{attribute addProperty BoxType "EK1122-0000-0018"}
{attribute addProperty Id "Beckhoff_EKM1xxxsub_EK1100EK1100_179A0949162A_0001_EKM1101_0000_0016EKM1101_87969BFD51464.25A_0002_EKM1101_0000_0017EKM1101_87969BFD51464.25A_0003_EKM1101_0000_0018EKM1101_87969BFD51464.25A_0004_EKM1101_0000_0019EKM1101_87969BFD51464.25A_0005_EKM1101_0000_0020EKM1101_87969BFD51464.25"}
{attribute addProperty CRC "2110049489"}
{attribute addProperty SizeInBites "2586"}
{attribute addProperty SizeInBytes "323.25"}
TYPE Beckhoff_EKM1xxxEK1122_7DC4CCD1 EXTENDS EK1122_179A0949 :
STRUCT
	{attribute addProperty Name "Beckhoff_EKM1xxxsub_EK1100"}
	Beckhoff_EKM1xxxsub_EK1100 : EK1100_179A0949;
	{attribute addProperty Name "A_0001_EKM1101_0000_0016"}
	A_0001_EKM1101_0000_0016 : EKM1101_87969BFD;
	{attribute addProperty Name "A_0002_EKM1101_0000_0017"}
	A_0002_EKM1101_0000_0017 : EKM1101_87969BFD;
	{attribute addProperty Name "A_0003_EKM1101_0000_0018"}
	A_0003_EKM1101_0000_0018 : EKM1101_87969BFD;
	{attribute addProperty Name "A_0004_EKM1101_0000_0019"}
	A_0004_EKM1101_0000_0019 : EKM1101_87969BFD;
	{attribute addProperty Name "A_0005_EKM1101_0000_0020"}
	A_0005_EKM1101_0000_0020 : EKM1101_87969BFD;
END_STRUCT
END_TYPE

(* stored: Version 1.2.0.0, ProductVersion 3.1.4024.9
   DUT Beckhoff_EKM1xxxEK1122_7DC4CCD1: Id {5478eba7-30df-4e83-82c3-2c9e84089863} *)
